Fanuc KAREL source: kd00071.KL

-- PROVISIONAL review KL for V1013-1; original PC SHA256 45dbb4ddfbf4cd78a00f7d48d6f1020e716e41e7c512494f646f58b1cd292063
-- Incomplete behavior may be omitted. Consult companion uncertainty JSON. Do not deploy.
PROGRAM KD00071
%NOLOCKGROUP
VAR
  I : INTEGER
  J : INTEGER
  B : BOOLEAN
  R : REAL
  S : STRING[80]
BEGIN
  -- UNRESOLVED_PC offsets 5-18; opcodes 9D,81,18,9D,1B,9D,12,9C,13,04
  -- UNRESOLVED_PC offsets 23-27; opcodes 7F
END KD00071
